FUNCTION_BLOCK RemoteAutoMng (* Basic Function Block Type *)
  (* Standard: 61499-2 *)
  (* Version 0.0, 6/3/2026, Schneider Electric, Template *)
  PACKAGE SE.Nereda;
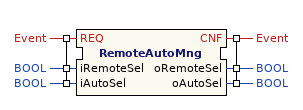
  EVENT_INPUT
    REQ WITH iRemoteSel, iAutoSel; (* Normal Execution Request *)
  END_EVENT
  EVENT_OUTPUT
    CNF WITH oRemoteSel, oAutoSel; (* Execution Confirmation *)
  END_EVENT
  VAR_INPUT
    iRemoteSel : BOOL;
    iAutoSel : BOOL;
  END_VAR
  VAR_OUTPUT
    oRemoteSel : BOOL;
    oAutoSel : BOOL;
  END_VAR
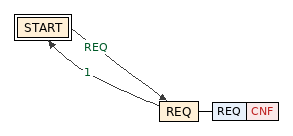
  EC_STATES
    START; (* Initial State *)
    REQ : REQ -> CNF; (* Normal execution *)
  END_STATES
  EC_TRANSITIONS
    START TO REQ := REQ;
    REQ TO START := 1;
  END_TRANSITIONS
  ALGORITHM REQ IN ST: (* Normally executed algorithm *)
;
IF iRemoteSel <> iAutoSel THEN
	oAutoSel := iAutoSel;
	oRemoteSel := iRemoteSel;
ELSE
	oAutoSel := FALSE;
	oRemoteSel := FALSE;
END_IF;
  END_ALGORITHM
END_FUNCTION_BLOCK
